// TIA Portal project "3M -5" (V16)

(* hardware
DEVICE "S7-1200 station_1"  S7-1200 Station
   slot 0: "Rack_0"  S7-1200 Rack  Rack  V1.0
   slot 1: "PLC_1"  CPU 1212C AC/DC/Rly  6ES7 212-1BE40-0XB0  V4.0
*)

// ===== PLC "PLC_1"  CPU 1212C AC/DC/Rly =====

VAR_GLOBAL   // PLC tag table "Default tag table"
   "K1" AT %Q0.0 : Bool;
   "stop1" AT %I0.4 : Bool;
   "k2" AT %Q0.1 : Bool;
   "X" AT %M0.2 : Bool;
   "K3" AT %Q0.2 : Bool;
   "start1" AT %I0.2 : Bool;
   "Tag_2" AT %M0.1 : Bool;
   "Tag_3" AT %M0.3 : Bool;
   "Tag_4" AT %M0.4 : Bool;
   "T5 tag" AT %M1.1 : Bool;
   "T4 tag" AT %M1.0 : Bool;
   "T1 tag" AT %M0.5 : Bool;
   "c1" AT %M3.0 : Bool;
   "C2" AT %M3.1 : Bool;
   "T2 tag" AT %M0.6 : Bool;
   "C3" AT %M3.2 : Bool;
   "T3 tag" AT %M0.7 : Bool;
   "C4" AT %M3.3 : Bool;
   "C5" AT %M3.4 : Bool;
   "STOP" AT %I0.3 : Bool;
END_VAR

// folder: System blocks/Program resources

DATA_BLOCK "T4"   // DB1
{ S7_Optimized_Access := 'TRUE' }
AUTHOR : Simatic
FAMILY : IEC
NAME : IEC_TMR
VERSION : 1.0
// stored: InstanceOfName IEC_TIMER
"IEC_TIMER"
BEGIN
END_DATA_BLOCK

DATA_BLOCK "T1"   // DB2
{ S7_Optimized_Access := 'TRUE' }
AUTHOR : Simatic
FAMILY : IEC
NAME : IEC_TMR
VERSION : 1.0
// stored: InstanceOfName IEC_TIMER
"IEC_TIMER"
BEGIN
END_DATA_BLOCK

DATA_BLOCK "T2"   // DB3
{ S7_Optimized_Access := 'TRUE' }
AUTHOR : Simatic
FAMILY : IEC
NAME : IEC_TMR
VERSION : 1.0
// stored: InstanceOfName IEC_TIMER
"IEC_TIMER"
BEGIN
END_DATA_BLOCK

DATA_BLOCK "T3"   // DB4
{ S7_Optimized_Access := 'TRUE' }
AUTHOR : Simatic
FAMILY : IEC
NAME : IEC_TMR
VERSION : 1.0
// stored: InstanceOfName IEC_TIMER
"IEC_TIMER"
BEGIN
END_DATA_BLOCK

DATA_BLOCK "T5"   // DB5
{ S7_Optimized_Access := 'TRUE' }
AUTHOR : Simatic
FAMILY : IEC
NAME : IEC_TMR
VERSION : 1.0
// stored: InstanceOfName IEC_TIMER
"IEC_TIMER"
BEGIN
END_DATA_BLOCK

// folder: (top level)

ORGANIZATION_BLOCK "Main"   // OB1, LAD, ProgramCycle
TITLE = "Main Program Sweep (Cycle)"
{ S7_Optimized_Access := 'TRUE' }
VERSION : 0.1
   VAR_INPUT
      Initial_Call : Bool;   // Initial call of this OB
      Remanence : Bool;   // =True, if remanent data are available
   END_VAR
BEGIN

REGION Network 1: start
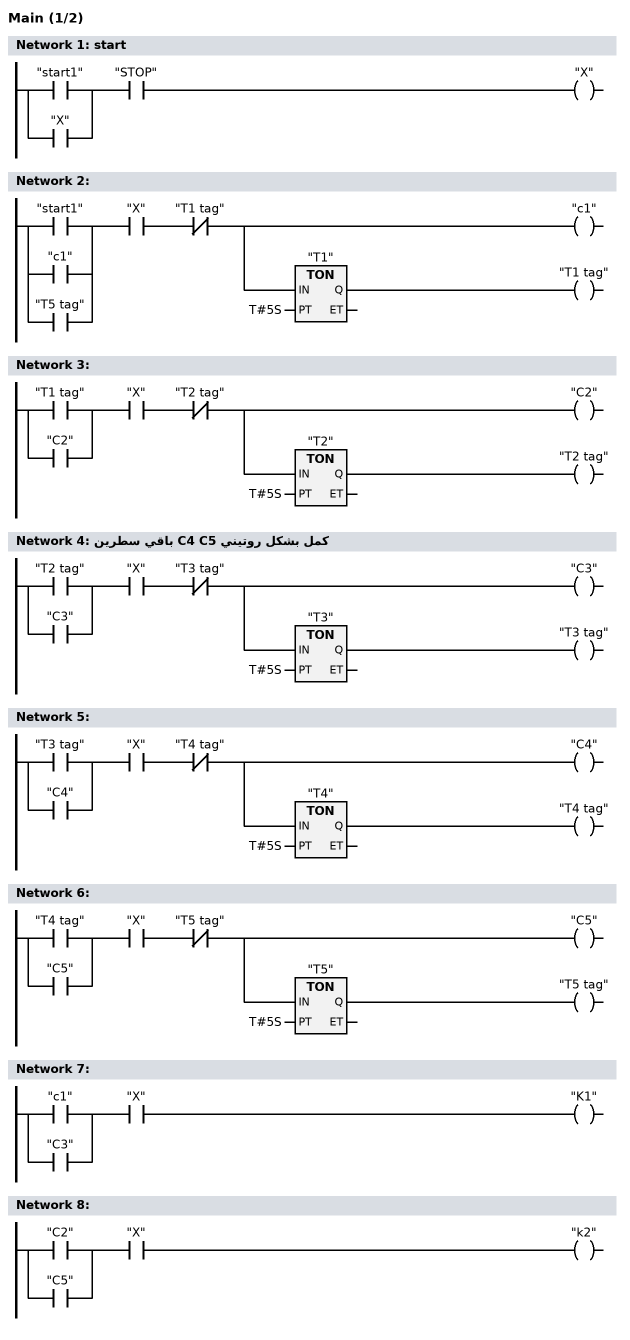
   RUNG wire#powerrail
      Contact( "start1" )
      wire#w1
      Contact( "STOP" )
      Coil( "X" )
   END_RUNG
   RUNG wire#powerrail
      Contact( "X" )
   END_RUNG wire#w1
   // the same network as SCL:
   "X" := ("start1" OR "X") AND "STOP";
END_REGION

REGION Network 2
   "c1" := ("start1" OR "c1" OR "T5 tag") AND "X" AND NOT "T1 tag";
   "T1".TON(IN := "c1", PT := T#5S);
   "T1 tag" := "T1".Q;
END_REGION

REGION Network 3
   "C2" := ("T1 tag" OR "C2") AND "X" AND NOT "T2 tag";
   "T2".TON(IN := "C2", PT := T#5S);
   "T2 tag" := "T2".Q;
END_REGION

REGION Network 4: باقي سطرين C4 C5 كمل بشكل روتيني
   "C3" := ("T2 tag" OR "C3") AND "X" AND NOT "T3 tag";
   "T3".TON(IN := "C3", PT := T#5S);
   "T3 tag" := "T3".Q;
END_REGION

REGION Network 5
   "C4" := ("T3 tag" OR "C4") AND "X" AND NOT "T4 tag";
   "T4".TON(IN := "C4", PT := T#5S);
   "T4 tag" := "T4".Q;
END_REGION

REGION Network 6
   "C5" := ("T4 tag" OR "C5") AND "X" AND NOT "T5 tag";
   "T5".TON(IN := "C5", PT := T#5S);
   "T5 tag" := "T5".Q;
END_REGION

REGION Network 7
   RUNG wire#powerrail
      Contact( "c1" )
      wire#w1
      Contact( "X" )
      Coil( "K1" )
   END_RUNG
   RUNG wire#powerrail
      Contact( "C3" )
   END_RUNG wire#w1
   // the same network as SCL:
   "K1" := ("c1" OR "C3") AND "X";
END_REGION

REGION Network 8
   RUNG wire#powerrail
      Contact( "C2" )
      wire#w1
      Contact( "X" )
      Coil( "k2" )
   END_RUNG
   RUNG wire#powerrail
      Contact( "C5" )
   END_RUNG wire#w1
   // the same network as SCL:
   "k2" := ("C2" OR "C5") AND "X";
END_REGION

REGION Network 9
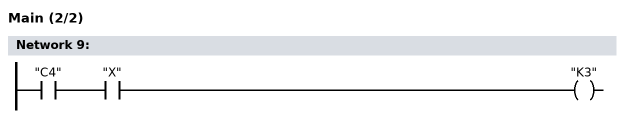
   RUNG wire#powerrail
      Contact( "C4" )
      Contact( "X" )
      Coil( "K3" )
   END_RUNG
   // the same network as SCL:
   "K3" := "C4" AND "X";
END_REGION
END_ORGANIZATION_BLOCK